TYPE ST_FlowControlParameters :
STRUCT
	movingAvgDurationSecs : INT;
	movingAvgShiftIntervalSecs : INT;
	co2ConsumptionLimit : DINT;
	excludeValuesPreFirstWindow : BOOL;
	startConsumptionCalculationWithAvg : BOOL;
END_STRUCT
END_TYPE

(* stored: Version 1.1.0.1, ProductVersion 3.1.4024.9
   DUT ST_FlowControlParameters: Id {59ca25a8-fcff-4997-971e-1b24e2fd5571} *)
